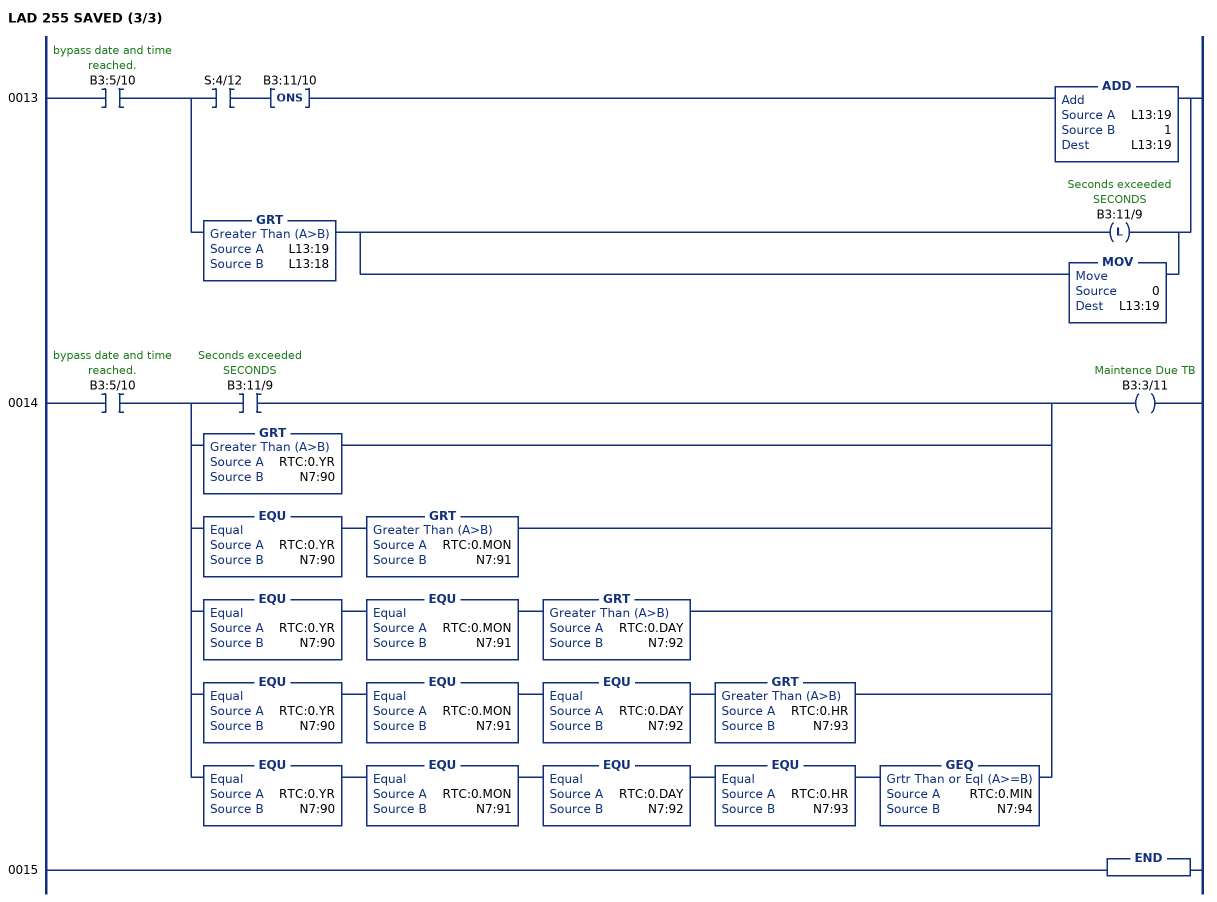
% Rung: 13 %
SOR XIC B3:5/10 BST XIC S:4/12 ONS B3:11/10 ADD L13:19 1 L13:19 NXB GRT L13:19 L13:18 BST OTL B3:11/9 NXB MOV 0 L13:19 BND BND EOR
%   B3:5/10  "bypass date and time reached." %
%   L13:18  MAX %
%   B3:11/9  SECONDS  "Seconds exceeded" %
% Rung: 14 %
SOR XIC B3:5/10 BST XIC B3:11/9 NXB GRT RTC:0.YR N7:90 NXB EQU RTC:0.YR N7:90 GRT RTC:0.MON N7:91 NXB EQU RTC:0.YR N7:90 EQU RTC:0.MON N7:91 GRT RTC:0.DAY N7:92 NXB EQU RTC:0.YR N7:90 EQU RTC:0.MON N7:91 EQU RTC:0.DAY N7:92 GRT RTC:0.HR N7:93 NXB EQU RTC:0.YR N7:90 EQU RTC:0.MON N7:91 EQU RTC:0.DAY N7:92 EQU RTC:0.HR N7:93 GEQ RTC:0.MIN N7:94 BND OTE B3:3/11 EOR
%   B3:5/10  "bypass date and time reached." %
%   B3:11/9  SECONDS  "Seconds exceeded" %
%   N7:90  RTC %
%   B3:3/11  TB  "Maintence Due" %
% Rung: 15 %
SOR END EOR

OTHER DOCUMENTED ADDRESSES
  B3:0/13  "toggle 2"
  B3:10/1  "bypass"
  B189:0/0  "change box"
  B189:0/9  "override boxing ok or not full signal"
  B189:0/11  "HMI force door close"
  B196:1/0  "Chute door is closed"
  B196:1/1  "control chute door"
  B196:1/13  "force box conveyor on"
  B196:3/0  "for hmi to continue production unlatched by hmi"
  HSC:0.0  "top"
  HSC:0.3/6  "Underflow interrupt"
  HSC:0.3/7  "Overflow interrupt"
  HSC:1.0  "bot"
  HSC:1.3/6  "Underflow interrupt"
  HSC:1.3/7  "Overflow interrupt"
  I:0.0/0  "Encoder Signal "A""
  I:0.0/1  "Encoder Signal "B""
  I:0.0/4  "Encoder Signal "A""
  I:0.0/5  "Encoder Signal "B""
  I:0.1/4  "not used"
  I:0.1/5  "not used"
  I:0.1/6  "not used"
  I:0.1/7  "not used"
  I:0.1/8  "not used"
  I:0.1/9  "not used"
  I:0.1/10  "not used"
  I:0.1/11  "not used"
  I:0.1/12  "not used"
  I:0.1/13  "not used"
  I:0.1/14  "not used"
  I:0.1/15  "not used"
  I:0.2  "not used"
  I:0.2/3  "Packaging Conveyor full"
  I:0.2/4  "Packaging Conveyor Box in Position"
  I:0.3  "not used"
  I:0.4  "Spare Analog Input 1"
  I:0.5  "Spare Analog Input 2"
  I:0.6  "Spare Analog Input 3"
  I:2.0/0  FRONT_ESTOP
  I:2.0/1  REAR_ESTOP
  I:2.0/8  FRONT_DOOR  "front door signal ce models only"
  I:2.0/9  REAR_DOOR  "rear door signal ce models only"
  I:2.0/11  "spare"
  L23:19  TOP_OPT_FAIL_CT
  L23:34  AIR_PRESSURE_FAULT
  L28:0  INS_1_TIME
  L29:0  INS_1_POS
  L30:0  INS_5_TIME
  L31:0  INS_5_POS
  L32:0  INS_6_TIME
  L33:0  INS_6_POS
  L192:1  BOT_LAST_TIME  "rtc bot belt previous movement event time"
  L192:2  BOT_CYCLE_TIME  "rtc bot belt time between events"
  L192:7  FROM_REAL  "distance from real part signal at optic location"
  L192:8  FROM_TRACKED  "distance from tracked part signal at optic location"
  L192:16  TOP_LAST_TIME  "rtc top belt previous movement event time"
  L192:17  TOP_CYCLE_TIME  "rtc top belt time between events"
  L199:5  ACQTM51
  L199:6  ACQTM52
  L199:7  ACQTM53
  L199:9  "ones"
  L199:10  "billions"
  L199:13  DUMP_LONG
  L199:15  ACQTM11
  L199:16  ACQTM12
  L199:17  ACQTM13
  L199:20  RESULTTM1
  L199:22  CLEARTIME5COUNT
  L199:23  CLEARTIME6COUNT
  L199:24  ACQTM61
  L199:25  ACQTM62
  L199:26  ACQTM63
  L199:27  TMSINCETRIG1
  L199:29  TMSINCETRIG5
  L199:30  TMSINCETRIG6
  L199:31  CLEARTIME1COUNT
  L199:32  RESULTTM5
  L199:33  RESULTTM6
  L199:34  MAXACQTM1
  L199:36  MAXACQTM6
  N7  
  N101:2  I3_TRIG_LOC
  N101:3  I4_TRIG_LOC
  O:0.0/1  "spare"
  O:0.0/11  "Spare"
  O:0.0/12  "not used"
  O:0.0/13  "not used"
  O:0.0/14  "not used"
  O:0.0/15  "not used"
  O:0.1  "not used"
  O:0.2  "not used"
  O:0.3  "not used"
  O:0.5  "spare analog output"
  O:3.0/0  "spare"
  O:3.0/2  "spare"
  O:3.0/3  "light curtain range selection /* needed? */"
  O:3.0/7  "door unlocks on CE models"
  O:3.0/8  "Light?"
  PFILE:6  "check for part jams"
  PFILE:10  "Bottom belt HSC"
  PFILE:12  "Top belt HSC"
  Q2:55  END_OF_MAIN
  Q5:94  END_OF_BELTS
  T20:0  "Trigger On Time"
  U:9  "slow data"
  U:24  "check skipped fail rate"
  U:28  "faults"
  U:29  "speed"
  U:30  "count"
  U:31  "rate calc"
  U:32  "boxer"
  U:33  "bulk pack"
  U:34  "customer boxing unit signals"
  U:35  "cleanup"

COMMENTS NOT ATTACHED TO A CURRENT RUNG
  R6:2: B41 is the top good 3 file
  R6:11/DN: B39 is the top good 2 file
  R6:10/DN: B37 is the top good 1 file
  R6:6/DN: B35 is the top NG file
  R6:0: B36 is the bottom GOOD file
  R6:4: B34 is the bottom NG file
  R6:6: B35 is the top NG file
  R6:10: B37 is the top good 1 file

REVISION NOTES
  13: updated count reset
  14: added io moduals
  15: multiple steps toward new hmi integration
  21: test
  27: fix error if bulk pack and no boxing fallout were on

DATA TABLE (non-zero values as saved)
DATA B3
% B3:0 % 0X8822 0X9141 0X4003 0XA101 0X0EBF 0X1540 0X15B8 0X0421 0X3F80 0X22D0
% B3:10 % 0X21FC 0X00CE 0X4000 0X8000 0X0000 0X0000 0X0000 0X0000 0X0000 0X0000
% B3:50 % 0X0001 0X0000 0X0000 0X0000 0X0000 0X0000 0X0000 0X0000 0X0000 0X0000
DATA T4
% .PRE .ACC %
% T4:0 % 0 1
% T4:1 % 150 0
% T4:2 % 400 0
% T4:3 % 500 147
% T4:4 % 1000 1000
% T4:5 % 5 5
% T4:6 % 10 32766
% T4:7 % 150 0
% T4:8 % 20 9
% T4:9 % 50 33
% T4:10 % 200 200
% T4:11 % 111 0
% T4:12 % 20 20
% T4:13 % 250 0
% T4:14 % 666 0
% T4:15 % 1000 1000
% T4:16 % 400 0
% T4:17 % 100 14
% T4:18 % 5 0
% T4:19 % 300 0
% T4:20 % 200 0
% T4:21 % 200 0
% T4:22 % 200 0
% T4:23 % 250 0
% T4:24 % 666 0
% T4:25 % 666 0
% T4:26 % 666 0
% T4:27 % 250 0
% T4:28 % 250 0
% T4:29 % 5000 0
% T4:30 % 333 142
% T4:31 % 500 142
% T4:32 % 500 144
% T4:33 % 500 141
DATA C5
% .PRE .ACC %
% C5:0 % 32766 0
DATA R6
% .LEN .POS %
% R6:0 % 1250 0
% R6:1 % 16 0
% R6:2 % 1050 0
% R6:3 % 1050 0
% R6:4 % 1250 0
% R6:5 % 1250 0
% R6:6 % 1713 0
% R6:7 % 16 0
% R6:8 % 1024 0
% R6:9 % 3 0
% R6:10 % 1713 0
% R6:11 % 1050 0
% R6:12 % 10 0
% R6:13 % 10 0
% R6:14 % 10 0
% R6:15 % 10 0
% R6:16 % 1713 0
% R6:17 % 1713 0
% R6:18 % 1050 0
% R6:19 % 10 0
DATA N7
% N7:0 % 17248 3 1125 300 3 0 0 0 500 43
% N7:10 % 1000 43 0 2 20 20 1000 2000 50 1050
% N7:20 % 0 1329 10 2000 222 46 0 0 0 250
% N7:30 % 666 1417 150 0 0 1221 76 25 0 25
% N7:40 % 3 29 0 29 32767 482 1217 1350 1636 1
% N7:50 % 0 16 1 16 17 1024 0 0 32766 3
% N7:60 % 1713 1713 1050 984 1034 1024 4999 5 400 400
% N7:70 % 100 200 300 400 90 190 290 390 16831 15891
% N7:80 % 0 0 1241 1246 1300 1310 13 26 0 0
% N7:90 % 2011 4 4 12 1 13 26 222 222 12
% N7:100 % 1003 90 110 100 175 25 0 0 0 0
% N7:190 % -128 27477 27605 32767 0 0 0 0 0 0
DATA F8
% F8:0 % 6
DATA L13
% L13:0 % 12164 115616 0 36352 171228
% L13:5 % 1309 5290 1309 141974 1113
% L13:10 % 1050 -2147483648 30832 15 90
% L13:15 % -1686106703 -2147483648 2147483647 2147483647 82058
% L13:20 % 67790938 -2111178937 777 34309 100
% L13:25 % 104 2245 -2147483648 1198 2096829497
% L13:30 % 512030702 1309 1020000 1572502331 444
% L13:35 % 0 11 99 912231227 912231260
% L13:40 % 0 1000000000 1000000 1572502304 -2028734845
% L13:45 % -2028734755 33 0 27 20163346
% L13:50 % 342628165 1842945 -2028735007 0 0
% L13:55 % 342628075 342628327 4936 0 -1783954972
% L13:60 % 26 104 -1783954986 600 -1
% L13:65 % 100 -100 -1787662150 912220637 12
% L13:70 % 2145981679 23 118 0 20163346
% L13:75 % 922236 60 100 -2028734984 1
% L13:80 % 24 74 74 7 493582
% L13:85 % 625579 56 0 0 342628200
% L13:90 % 342628110 5 36041 5 2096849366
% L13:95 % 10 256 0 -2028734724 89425
% L13:100 % 182972200 6 3000 14 169383001
% L13:105 % 89425 31 59896194 9157696 59896188
% L13:110 % 6 100 50 2117450677 -2111804757
% L13:115 % -2111804511 246 123 -2111804634 26
% L13:120 % 5 -2147483648 50 100 10
% L13:125 % 0 2145981679 2147483647 3276500 66337692
% L13:130 % 2 2 0 99 0
% L13:135 % 0 0 625584 5 70
% L13:140 % 0 5 36 50 50
% L13:145 % 1843080 5 5 5 11
% L13:150 % 12 20 1263072 -1263072 2147483647
% L13:155 % 0 -10 0 0 4589052
% L13:160 % 6 27 31 1220 45
% L13:165 % 2119507177 2145981707 2119507177 2145981707 6706
% L13:170 % 12817 169383112 169383174 400 2400
% L13:175 % 4 4 42 23 38
% L13:180 % -1787662150 0 0 1000000 0
% L13:185 % 0 0 912245139 27 50951
% L13:190 % 56000000 0 0 0 0
DATA L19
% L19:0 % -2028736811 2096829497 2096829921 2096830067 2096830267
% L19:5 % 2096830448 2096830689 2096831120 2096831297 2096831585
% L19:10 % 2096833666 2096836638 2096837135 2096840674 2096842366
% L19:15 % 2096842953 2096848724 0 0 0
DATA L20
% L20:0 % 2096830885 2096831065 2096831307 2096831737 2096831912
% L20:5 % 2096832202 2096834281 2096837255 2096837751 2096841293
% L20:10 % 2096842979 2096843569 2096849339 -2028734845 2093033638
% L20:15 % 2093033777 2093033948 2093034392 2096791590 2096791726
% L20:20 % 2096791887 2096792035 2096792316 2096792630 2096792846
% L20:25 % 2096793019 2096793171 2096793313 2096793506 2096793755
% L20:30 % 2096794012 2096794203 2096794410 2096810455 2096810591
% L20:35 % 2096810710 2096810849 2096811036 2096811809 2096828656
% L20:40 % 2096828818 2096828917 2096829019 2096829127 2096829230
% L20:45 % 2096829388 2096829705 2096830114 2096830539 2096830683
DATA L21
% L21:0 % 2119500665 2119500729 2119500814 2119500966 2119501028
% L21:5 % 2119501130 2119501864 2119502913 2119503088 2119504337
% L21:10 % 2119504933 2119505141 2119507177 2145981697 2118160917
% L21:15 % 2118160966 2118161026 2118161183 2119486802 2119486850
% L21:20 % 2119486907 2119486959 2119487058 2119487169 2119487245
% L21:25 % 2119487306 2119487360 2119487410 2119487478 2119487566
% L21:30 % 2119487657 2119487724 2119487797 2119493458 2119493506
% L21:35 % 2119493548 2119493597 2119493663 2119493936 2119499879
% L21:40 % 2119499936 2119499971 2119500007 2119500045 2119500081
% L21:45 % 2119500137 2119500249 2119500393 2119500543 2119500594
DATA L22
% L22:0 % 2096811064 2096811837 2096828684 2096828846 2096828945
% L22:5 % 2096829047 2096829156 2096829258 2096829416 2096829733
% L22:10 % 2096830142 2096830567 2096830711 2096830913 2096831094
% L22:15 % 2096831335 2096831765 2096831941 2096832230 2096834310
% L22:20 % 2096837283 2096837779 2096841321 2096843008 2096843597
% L22:25 % 2096849367 -2028734755 2093033666 2093033806 2093033976
% L22:30 % 2093034420 2096791618 2096791754 2096791916 2096792063
% L22:35 % 2096792344 2096792658 2096792874 2096793046 2096793199
% L22:40 % 2096793341 2096793534 2096793784 2096794041 2096794231
% L22:45 % 2096794439 2096810483 2096810619 2096810738 2096810878
DATA L23
% L23:0 % 2119493673 2119493946 2119499889 2119499946 2119499981
% L23:5 % 2119500017 2119500055 2119500091 2119500147 2119500259
% L23:10 % 2119500403 2119500553 2119500604 2119500675 2119500739
% L23:15 % 2119500824 2119500976 2119501038 2119501140 2119501874
% L23:20 % 2119502923 2119503098 2119504347 2119504943 2119505151
% L23:25 % 2119507187 2145981707 2118160927 2118160976 2118161036
% L23:30 % 2118161193 2119486812 2119486860 2119486917 2119486969
% L23:35 % 2119487068 2119487179 2119487255 2119487316 2119487370
% L23:40 % 2119487420 2119487488 2119487576 2119487667 2119487734
% L23:45 % 2119487807 2119493468 2119493516 2119493558 2119493607
DATA L30
% L30:0 % 1097513510 1097513738 1097513967 1097514196 1097514426
% L30:5 % 1097514655 1097514883 1097515111 1097515339 1569237509
% L30:10 % 1571789345 1571789602 1571790886 1571791144 1571791400
% L30:15 % 1572418698 1572420630 1572420885 1572422166 1572422422
% L30:20 % 1572422681 1572500242 1572500500 1572501791 1572502048
% L30:25 % 1572502304 1071308573 1071308799 1071309024 1071309250
% L30:30 % 1071309476 1071429569 1071429795 1071431153 1071431379
% L30:35 % 1071431606 1088333039 1088333266 1088334623 1088334848
% L30:40 % 1088335075 1089808842 1089809070 1089810430 1089810657
% L30:45 % 1089810882 1092780028 1092791426 1092806921 1097513283
DATA L31
% L31:0 % 3522828 3522897 3522967 3523035 3523105
% L31:5 % 3523175 3523244 3523313 3523382 18677621
% L31:10 % 19955820 19955950 19956596 19956726 19956855
% L31:15 % 20121868 20122368 20122448 20122938 20123054
% L31:20 % 20123174 20162306 20162436 20163087 20163217
% L31:25 % 20163346 2077757 2077757 2077757 2077757
% L31:30 % 2077757 2077757 2077757 2077757 2077757
% L31:35 % 2077757 2077757 2077757 2077757 2077757
% L31:40 % 2077757 2077757 2077757 2077757 2077757
% L31:45 % 2077757 2091375 2094821 2099507 3522760
DATA L32
% L32:0 % 2096810540 2096810659 2096810798 2096810985 2096811758
% L32:5 % 2096828605 2096828767 2096828865 2096828968 2096829075
% L32:10 % 2096829179 2096829337 2096829654 2096830063 2096830488
% L32:15 % 2096830632 2096830833 2096831015 2096831255 2096831686
% L32:20 % 2096831862 2096832151 2096834230 2096837203 2096837700
% L32:25 % 2096841242 2096842929 2096843518 2096849288 -2028735007
% L32:30 % 2093033586 2093033726 2093033897 2093034341 2096791539
% L32:35 % 2096791674 2096791836 2096791984 2096792265 2096792579
% L32:40 % 2096792794 2096792968 2096793120 2096793261 2096793455
% L32:45 % 2096793704 2096793962 2096794152 2096794359 2096810404
DATA L33
% L33:0 % 2119493488 2119493530 2119493579 2119493645 2119493918
% L33:5 % 2119499861 2119499918 2119499953 2119499989 2119500027
% L33:10 % 2119500063 2119500119 2119500231 2119500375 2119500525
% L33:15 % 2119500576 2119500647 2119500711 2119500796 2119500948
% L33:20 % 2119501010 2119501112 2119501846 2119502895 2119503070
% L33:25 % 2119504319 2119504915 2119505123 2119507159 2145981679
% L33:30 % 2118160899 2118160948 2118161008 2118161165 2119486784
% L33:35 % 2119486832 2119486889 2119486941 2119487040 2119487151
% L33:40 % 2119487227 2119487288 2119487342 2119487392 2119487460
% L33:45 % 2119487548 2119487639 2119487706 2119487779 2119493440
DATA B40
% B40:0 % 0XAAAA
DATA B100
% B100:0 % 0X3700 0X18A8 0X000C 0X0000 0X0000 0X0000 0X0000 0X0000 0X0000 0X0000
DATA N101
% N101:0 % 118 16383 0 0 1183 100 1002 1200 1212 1230
% N101:10 % 1240 1632 10 16383 1024 0 3000 500 333 500
% N101:20 % 1000 500 400 0 0 0 500 500 0 0
DATA L102
% L102:0 % 20 10 1 1102 0
% L102:5 % 1100 0 0 0 0
% L102:10 % 0 727 1 1 36041
% L102:15 % 0 30 10 40 10
% L102:20 % 17 4 69362 0 27
% L102:25 % 27 0 1829722 81649 714735
% L102:30 % 23 5 30 7754 0
% L102:35 % 0 50 0 999999 31
% L102:40 % 14 24 63160 0 0
